// TIA Portal V17 export
// export: Created 2022-03-10T13:08:27.0782031Z, ExportSetting WithDefaults, DisplayName Totally Integrated Automation Portal, DisplayVersion V17, DisplayName TIA Portal Openness, DisplayVersion V17, DisplayName TIA Portal Teamcenter Gateway, DisplayVersion V17, DisplayName TIA Portal Version Control Interface, DisplayVersion V17, DisplayName SINAMICS Startdrive Advanced, DisplayVersion V17, DisplayName SINAMICS Startdrive G130, G150, S120, S150, SINAMICS MV, S210, DisplayVersion V17, DisplayName SINAMICS Startdrive G110M, G120, G120C, G120D, G120P, G115D, DisplayVersion V17, DisplayName STEP 7 Professional, DisplayVersion V17, DisplayName STEP 7 Safety, DisplayVersion V17, DisplayName WinCC Advanced / Unified PC, DisplayVersion V17
FUNCTION_BLOCK "fbAlarmesFalhas"   // FB5, LAD
{ S7_Optimized_Access := 'TRUE' }
VERSION : 0.1
// stored: AutoNumber false, IsIECCheckEnabled false, SetENOAutomatically false, UDAEnableTagReadback false
   VAR
      xAlarmesOk : Array[0..7] of Bool;
      xFalhasOk : Array[0..7] of Bool;
      xEmergenciaOk : Array[0..7] of Bool;
      xResetGeral : Bool;
   END_VAR
BEGIN

REGION Network 1: Sistema de Segurança / Emergência
END_REGION

REGION Network 2: Disjuntores
END_REGION

REGION Network 3: Drives e Motores / Processo
END_REGION

REGION Network 4: ------------------------------------------------------Gerenciamento----------------------------------------------------- / ================== Gerenciamento de Status ==================
END_REGION

REGION Network 5: Emergência OK / Emergência Ok
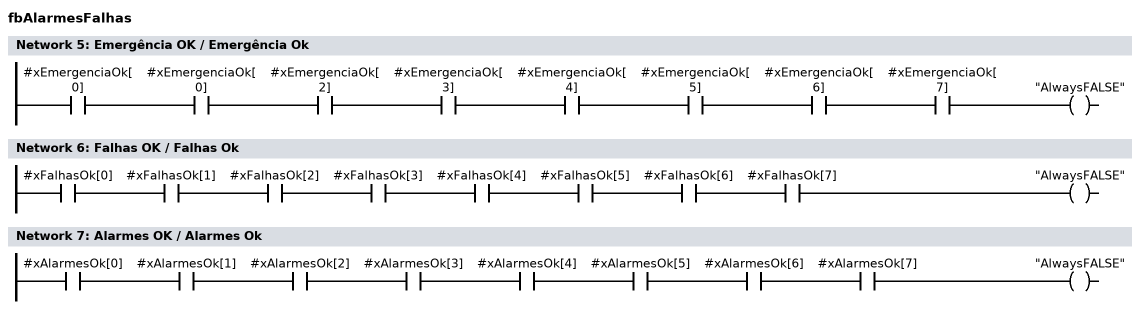
   RUNG wire#powerrail
      Contact( #xEmergenciaOk[0] )
      Contact( #xEmergenciaOk[0] )
      Contact( #xEmergenciaOk[2] )
      Contact( #xEmergenciaOk[3] )
      Contact( #xEmergenciaOk[4] )
      Contact( #xEmergenciaOk[5] )
      Contact( #xEmergenciaOk[6] )
      Contact( #xEmergenciaOk[7] )
      Coil( "AlwaysFALSE" )
   END_RUNG
   // the same network as SCL:
   "AlwaysFALSE" := #xEmergenciaOk[0] AND #xEmergenciaOk[0] AND #xEmergenciaOk[2] AND #xEmergenciaOk[3] AND #xEmergenciaOk[4] AND #xEmergenciaOk[5] AND #xEmergenciaOk[6] AND #xEmergenciaOk[7];
END_REGION

REGION Network 6: Falhas OK / Falhas Ok
   RUNG wire#powerrail
      Contact( #xFalhasOk[0] )
      Contact( #xFalhasOk[1] )
      Contact( #xFalhasOk[2] )
      Contact( #xFalhasOk[3] )
      Contact( #xFalhasOk[4] )
      Contact( #xFalhasOk[5] )
      Contact( #xFalhasOk[6] )
      Contact( #xFalhasOk[7] )
      Coil( "AlwaysFALSE" )
   END_RUNG
   // the same network as SCL:
   "AlwaysFALSE" := #xFalhasOk[0] AND #xFalhasOk[1] AND #xFalhasOk[2] AND #xFalhasOk[3] AND #xFalhasOk[4] AND #xFalhasOk[5] AND #xFalhasOk[6] AND #xFalhasOk[7];
END_REGION

REGION Network 7: Alarmes OK / Alarmes Ok
   RUNG wire#powerrail
      Contact( #xAlarmesOk[0] )
      Contact( #xAlarmesOk[1] )
      Contact( #xAlarmesOk[2] )
      Contact( #xAlarmesOk[3] )
      Contact( #xAlarmesOk[4] )
      Contact( #xAlarmesOk[5] )
      Contact( #xAlarmesOk[6] )
      Contact( #xAlarmesOk[7] )
      Coil( "AlwaysFALSE" )
   END_RUNG
   // the same network as SCL:
   "AlwaysFALSE" := #xAlarmesOk[0] AND #xAlarmesOk[1] AND #xAlarmesOk[2] AND #xAlarmesOk[3] AND #xAlarmesOk[4] AND #xAlarmesOk[5] AND #xAlarmesOk[6] AND #xAlarmesOk[7];
END_REGION
END_FUNCTION_BLOCK
